// TIA Portal V19 export
FUNCTION "M_CmpLTE" : Bool   // FC14, LAD
TITLE = Module compare LOWER THAN EQUAL / Module compare Lower than equal
// stored: Access Published, SetENOAutomatically false
   VAR_INPUT
      Xa : LReal;
      Xb : LReal;
      MODULE : LReal;
   END_VAR
BEGIN

REGION Network 1 (SCL): Xa <= Xb return TRUE / Main
   #M_CmpLTE := "M_PosAMinusPosB"(PosA := #Xa, PosB := #Xb, MODULE := #MODULE) <= 0.0;
END_REGION
END_FUNCTION
